// TIA Portal V18 export
DATA_BLOCK "H-8_PID"   // DB70
{ S7_Optimized_Access := 'TRUE' }
VERSION : 0.1
// stored: AutoNumber true, DBAccessibleFromOPCUA true, DBAccessibleFromWebserver true, IsOnlyStoredInLoadMemory false, IsRetainMemResEnabled false, IsWriteProtectedInAS false, MemoryReserve 100
   VAR RETAIN
      Data { S7_SetPoint := 'True'} : "PID_DT";
   END_VAR
BEGIN
   Data.k := 1.2;
   Data.Ti := T#2S;
   Data.ManualInput := 37.16286;
   Data.OutPutValue := 37.16286;
   Data.OutPutMin := 10.0;
   Data.OutPutMax := 45.0;
   Data.Control := 16#0000;
   Data.SP1 := 1.3;
   Data.SP2 := 0.0;
   Data.SP3 := 0.0;
   Data.SP4 := 0.0;
   Data.SP5 := 0.0;
   Data.SPActive := 1.3;
END_DATA_BLOCK
